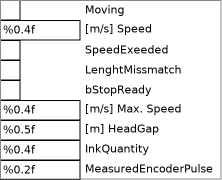
VISUALIZATION _VISU_Pm_MachineOut  // 222x180
VAR_IN_OUT
	ref : ST_ModuleMachineInterface_OUT;
END_VAR
    Rectangle (0,20 80x20), "%0.4f", text variable: ref.fSpeed
    Rectangle (82,20 140x18), "[m/s] Speed"
    Rectangle (0,100 80x20), "%0.4f", text variable: ref.fMaxSpeed
    Rectangle (82,100 140x18), "[m/s] Max. Speed"
    Rectangle (82,0 140x20), "Moving"
    RoundedRectangle (0,40 20x20), colour toggle: ref.bSpeedExeeded
    Rectangle (82,40 140x20), "SpeedExeeded"
    RoundedRectangle (0,0 20x20), colour toggle: ref.bMoving
    Rectangle (0,120 80x20), "%0.5f", text variable: ref.fHeadGap
    Rectangle (82,120 140x18), "[m] HeadGap"
    Rectangle (0,140 80x20), "%0.4f", text variable: ref.fInkQuantity
    Rectangle (82,140 140x18), "InkQuantity"
    Rectangle (0,160 80x20), "%0.2f", text variable: ref.fEncoderStepsMeasured
    Rectangle (82,160 140x18), "MeasuredEncoderPulse"
    RoundedRectangle (0,60 20x20), colour toggle: ref.bLengthMismatch
    Rectangle (82,60 140x20), "LenghtMissmatch"
    RoundedRectangle (0,80 20x20), colour toggle: ref.bStopReady
    Rectangle (82,80 140x20), "bStopReady"
END_VISUALIZATION

(* stored: Version 1.1.0.1, ProductVersion 3.1.4024.11
   Visu _VISU_Pm_MachineOut: Id {7baff7a3-f273-4514-85b8-8e939f801947} *)
